PROGRAM FirstApp
VAR
	bIN: BOOL;
	bOut: BOOL;
	bIn2: BOOL;
END_VAR

bOut := NOT bIN AND bIn2;

END_PROGRAM

(* stored: Version 1.1.0.1, ProductVersion 3.1.4024.11
   POU FirstApp: Id {a16bda55-b8de-441b-a22b-d088f2e9b3a9}, SpecialFunc None *)
